ABB RobotStudio station: IRB_drawing_interface.rspag

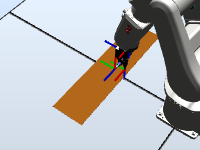
--- station ---
Station IRB_drawing_interface (saved by RobotStudio 6.7.7985.1011)
Controller IRB_120_3kg_0.58m
  mechanical unit ROB_1: IRB120_3_58__01, 6 joints, base frame (0, 0, 0) mm
Layout (positions relative to the parent item):
  - IRB120_3_58__01 [mechanism, from Robots\IRB120_3_58_G_01.rslib] at (0, 0, 0) mm; joint values [-0.0847, 0.5499, 0.7011, 0, 0.3197, 1.4861] (rad or m)
  - writing_tool_v3.1 [mechanism, from Libraries\writing_tool_v3.1.rslib] at (301.4, -25.6, 183.5) mm, rotated rx 180 ry 0 rz 90 deg
  - Cylinder_150_75_40_140_r47 [part] at (0, 0, 14) mm
  - Surface_600_150 [part]
Attachment: writing_tool_v3.1 is attached to IRB120_3_58__01 / Link6

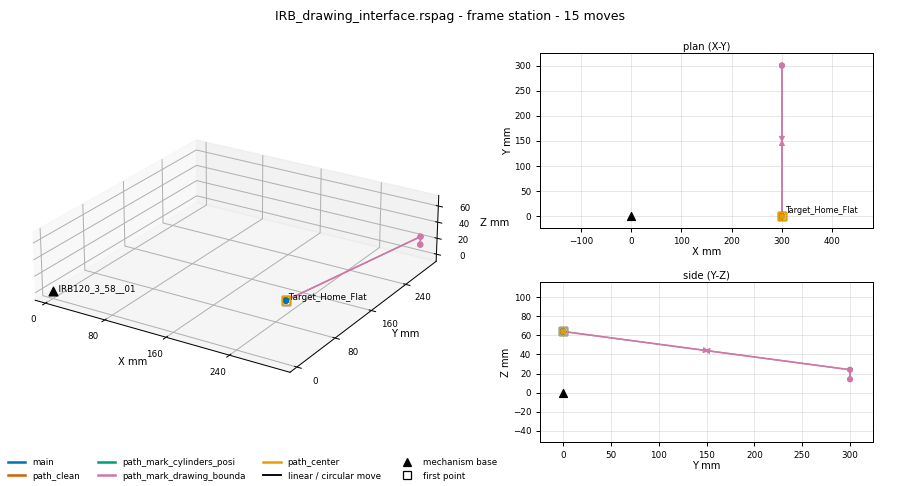
[picture p0: tool path of IRB_drawing_interface.rspag in frame station, 15 of 55 moves have a stored position in this frame; points joined in program order, loops and branches not executed]
--- Backups/IRB_120_3kg_0.58m/RAPID/TASK1/PROGMOD/Module1.mod ---
MODULE Module1

    CONST num default_flat_surface_width := 600;
    CONST num default_flat_surface_height := 150;
    CONST num default_cylinder_center_x:= 150;
    CONST num default_cylinder_center_y:=75;
    CONST num default_cylinder_bottom_height := 40;
    CONST num default_cylinder_top_height := 140;
    CONST num default_cylinder_radius := 47;

    CONST num default_cylinder_clearance := 10;
    CONST num default_cleaning_clearance := 20;

    VAR bool flag_flat:=TRUE;
    VAR bool flag_cylinder:=FALSE;
    VAR bool flag_change := TRUE;

    VAR pos message_target_pos;
    VAR intnum connectnum_pos;
    VAR string message_string;
    VAR intnum connectnum_string;

    VAR pos targetList{50000};
    VAR num targetListCount:=1;
    VAR num currentTarget:=1;

    VAR bool clean_writing_area:=FALSE;
    VAR bool stop_writing := FALSE;
    VAR bool center_the_cylinder := FALSE;
    VAR bool mark_cylinders_position := FALSE;
    VAR bool mark_drawing_boundaries := FALSE;

    VAR num flat_surface_width := default_flat_surface_width;
    VAR num flat_surface_height := default_flat_surface_height;
    VAR num cylinder_center_x:= default_cylinder_center_x;
    VAR num cylinder_center_y:=default_cylinder_center_y;
    VAR num cylinder_bottom_height := default_cylinder_bottom_height;
    VAR num cylinder_top_height := default_cylinder_top_height;
    VAR num cylinder_radius := default_cylinder_radius;
    VAR num angle;
    VAR pos flat_current_point := [0,0,47 + default_cylinder_clearance];
    VAR num cylinder_start_angle := 0;

	PERS tooldata side:=[TRUE,[[70.1,18.6,86],[0.707106781,0,0.707106781,0]],[0.4,[0,0,50],[1,0,0,0],0,0,0]];
	PERS tooldata down:=[TRUE,[[25.6,-1.4,119.5],[1,0,0,0]],[0.4,[0,0,50],[1,0,0,0],0,0,0]];
	PERS tooldata clean:=[TRUE,[[2.6,46.6,43],[0.5,-0.5,0.5,0.5]],[0.4,[0,0,50],[1,0,0,0],0,0,0]];

	PERS wobjdata WritingArea:=[FALSE,TRUE,"",[[300,300,14],[0.707,0,0,-0.707]],[[0,0,0],[1,0,0,0]]];

    CONST robtarget Target_Home_Flat:=[[300,0,50],[0,0,1,0],[0,-1,-1,0],[9E+09,9E+09,9E+09,9E+09,9E+09,9E+09]];
    VAR robtarget Target_Home_Cylinder:=[[150+default_cylinder_radius+default_cylinder_clearance,default_cylinder_center_y,default_cylinder_bottom_height],[0.707,0,-0.707,0],[0,-1,-1,0],[9E+09,9E+09,9E+09,9E+09,9E+09,9E+09]];
    CONST robtarget cleaning_target_1 := [[15,0,default_cleaning_clearance],[0,0.707,-0.707,0],[0,0,-2,1],[9E+09,9E+09,9E+09,9E+09,9E+09,9E+09]];
    CONST robtarget cleaning_target_2 := [[15,0,default_cleaning_clearance],[0,-1,.000191058,0],[0,-1,-2,1],[9E+09,9E+09,9E+09,9E+09,9E+09,9E+09]];

    PROC main()

        CONNECT connectnum_pos WITH RABMsgs_pos;
        IRMQMessage message_target_pos,connectnum_pos;
        CONNECT connectnum_string WITH RABMsgs_string;
        IRMQMessage message_string,connectnum_string;

        WHILE flag_flat=TRUE DO

            IF stop_writing THEN
                currentTarget := targetListCount;
                stop_writing := FALSE;

            ELSEIF flag_change THEN
                MoveL Target_Home_Flat,v300,z10,down\WObj:=WritingArea;
                flag_change := FALSE;

            ELSEIF clean_writing_area THEN
                path_clean;
                clean_writing_area := FALSE;

            ELSEIF center_the_cylinder THEN
                path_center;
                center_the_cylinder := FALSE;

            ELSEIF mark_cylinders_position THEN
                path_mark_cylinders_position;
                mark_cylinders_position := FALSE;

            ELSEIF mark_drawing_boundaries THEN
                path_mark_drawing_boundaries;
                mark_drawing_boundaries := FALSE;

            ELSEIF (currentTarget<>targetListCount) THEN

                targetList{currentTarget}.y:= -1 * targetList{currentTarget}.y + flat_surface_height;

                IF targetList{currentTarget}.z=0 THEN
                    MoveJ [[targetList{currentTarget}.x,targetList{currentTarget}.y,targetList{currentTarget}.z+10],[0,0,1,0],[0,-1,-1,0],[9E+09,9E+09,9E+09,9E+09,9E+09,9E+09]],v200,z10,down\WObj:=WritingArea;
                    MoveL [[targetList{currentTarget}.x,targetList{currentTarget}.y,targetList{currentTarget}.z],[0,0,1,0],[0,-1,-1,0],[9E+09,9E+09,9E+09,9E+09,9E+09,9E+09]],v300,fine,down\WObj:=WritingArea;
                ELSEIF targetList{currentTarget}.z=1 THEN
                    MoveL [[targetList{currentTarget}.x,targetList{currentTarget}.y,targetList{currentTarget}.z],[0,0,1,0],[0,-1,-1,0],[9E+09,9E+09,9E+09,9E+09,9E+09,9E+09]],v300,fine,down\WObj:=WritingArea;
                ELSEIF targetList{currentTarget}.z=2 THEN
                    MoveL [[targetList{currentTarget}.x,targetList{currentTarget}.y,targetList{currentTarget}.z],[0,0,1,0],[0,-1,-1,0],[9E+09,9E+09,9E+09,9E+09,9E+09,9E+09]],v300,fine,down\WObj:=WritingArea;
                    MoveJ [[targetList{currentTarget}.x,targetList{currentTarget}.y,targetList{currentTarget}.z+10],[0,0,1,0],[0,-1,-1,0],[9E+09,9E+09,9E+09,9E+09,9E+09,9E+09]],v200,z10,down\WObj:=WritingArea;
                ENDIF
                currentTarget:=currentTarget+1;

            ELSE
                MoveL Target_Home_Flat,v300,z10,down\WObj:=WritingArea;
            ENDIF

        ENDWHILE

        WHILE flag_cylinder=TRUE DO

            IF stop_writing THEN
                currentTarget := targetListCount;
                stop_writing := FALSE;

            ELSEIF flag_change THEN
                MoveL Target_Home_Flat,v300,z10,down\WObj:=WritingArea;
                MoveL Target_Home_Cylinder,v300,z10,side\WObj:=WritingArea;
                flag_change := FALSE;

            ELSEIF (currentTarget<>targetListCount) THEN

                targetList{currentTarget}.y:= -1 * targetList{currentTarget}.y + cylinder_top_height - cylinder_bottom_height;

                IF targetList{currentTarget}.z=0 THEN
                    curve_to_point([targetList{currentTarget}.x,targetList{currentTarget}.y, cylinder_radius + default_cylinder_clearance]);
                    curve_to_point([targetList{currentTarget}.x,targetList{currentTarget}.y, cylinder_radius]);
                ELSEIF targetList{currentTarget}.z=1 THEN
                    curve_to_point([targetList{currentTarget}.x,targetList{currentTarget}.y, cylinder_radius]);
                ELSEIF targetList{currentTarget}.z=2 THEN
                    curve_to_point([targetList{currentTarget}.x,targetList{currentTarget}.y, cylinder_radius]);
                    curve_to_point([targetList{currentTarget}.x,targetList{currentTarget}.y, cylinder_radius + default_cylinder_clearance]);
                ENDIF
                currentTarget:=currentTarget+1;

            ELSEIF clean_writing_area THEN
                !path_clean;
                clean_writing_area := FALSE;
            ELSE
                curve_to_point([0,0,cylinder_radius + default_cylinder_clearance]);
            ENDIF

        ENDWHILE

        IDelete connectnum_pos;
        IDelete connectnum_string;

    ENDPROC

    TRAP RABMsgs_pos

        VAR rmqmessage msg;
        VAR rmqheader header;
        VAR rmqslot rabclient;
        VAR num userdef;
        RMQGetMessage msg;
        RMQGetMsgHeader msg\Header:=header\SenderId:=rabclient\UserDef:=userdef;

        IF header.datatype="pos" THEN
            RMQGetMsgData msg,message_target_pos;

            targetList{targetListCount}:=message_target_pos;
            targetListCount:=targetListCount+1;

        ENDIF

    ENDTRAP

    TRAP RABMsgs_string

        VAR rmqmessage msg;
        VAR rmqheader header;
        VAR rmqslot rabclient;
        VAR num userdef;
        VAR num n;
        VAR num m;
        VAR bool convert_ok;
        RMQGetMessage msg;
        RMQGetMsgHeader msg\Header:=header\SenderId:=rabclient\UserDef:=userdef;

        IF header.datatype="string" THEN
            RMQGetMsgData msg,message_string;

            IF StrPart(message_string, 1, 4) = "func" THEN

                IF StrPart(message_string, 6, 1) = "1" THEN
                    stop_writing := TRUE;
                ELSEIF StrPart(message_string, 6, 1) = "2" THEN
                    clean_writing_area := TRUE;
                ELSEIF StrPart(message_string, 6, 1) = "3" THEN

                ELSEIF StrPart(message_string, 6, 1) = "4" THEN

                ELSEIF StrPart(message_string, 6, 1) = "5" THEN
                    center_the_cylinder := TRUE;
                ELSEIF StrPart(message_string, 6, 1) = "6" THEN
                    mark_cylinders_position := TRUE;
                ELSEIF StrPart(message_string, 6, 1) = "7" THEN
                    mark_drawing_boundaries := TRUE;
                ENDIF

            ELSEIF StrPart(message_string, 1, 4) = "para" THEN

                n := StrMatch(message_string, 1, "fsw");
                m := StrFind(message_string,n + 3,STR_WHITE);
                convert_ok := StrToVal(StrPart(message_string, n + 3, m - (n + 3)), flat_surface_width);

                n := StrMatch(message_string, 1, "fsh");
                m := StrFind(message_string,n + 3,STR_WHITE);
                convert_ok := StrToVal(StrPart(message_string, n + 3, m - (n + 3)), flat_surface_height);

                n := StrMatch(message_string, 1, "cpx");
                m := StrFind(message_string,n + 3,STR_WHITE);
                convert_ok := StrToVal(StrPart(message_string, n + 3, m - (n + 3)), cylinder_center_x);

                n := StrMatch(message_string, 1, "cpy");
                m := StrFind(message_string,n + 3,STR_WHITE);
                convert_ok := StrToVal(StrPart(message_string, n + 3, m - (n + 3)), cylinder_center_y);

                n := StrMatch(message_string, 1, "cbh");
                m := StrFind(message_string,n + 3,STR_WHITE);
                convert_ok := StrToVal(StrPart(message_string, n + 3, m - (n + 3)), cylinder_bottom_height);

                n := StrMatch(message_string, 1, "cth");
                m := StrFind(message_string,n + 3,STR_WHITE);
                convert_ok := StrToVal(StrPart(message_string, n + 3, m - (n + 3)), cylinder_top_height);

                n := StrMatch(message_string, 1, "cra");
                m := StrFind(message_string,n + 3,STR_WHITE);
                convert_ok := StrToVal(StrPart(message_string, n + 3, m - (n + 3)), cylinder_radius);

                n := StrMatch(message_string, 1, "cld");
                m := StrFind(message_string,n + 3,STR_WHITE);
                IF StrPart(message_string, n + 3, m - (n + 3)) = "True" THEN
                    flag_flat := FALSE;
                    flag_cylinder := TRUE;
                    flag_change := TRUE;
                ELSE
                    flag_flat := TRUE;
                    flag_cylinder := FALSE;
                    flag_change := TRUE;
                ENDIF

                Target_Home_Cylinder.trans := [150+cylinder_radius+default_cylinder_clearance,cylinder_center_y,cylinder_bottom_height];

            ENDIF
        ENDIF

    ENDTRAP

    PROC path_clean()
        CONST num cleaning_step := 52;
        VAR speeddata cleaning_speed := v200;
        VAR num offset_x := cleaning_step / 2;

        MoveJ Offs(Target_Home_Flat,0,0,0),cleaning_speed,z10,down\WObj:=WritingArea;
        MoveJ Offs(cleaning_target_1,cleaning_step / 2,flat_surface_height,120),cleaning_speed,z10,clean\WObj:=WritingArea;
        MoveJ Offs(cleaning_target_1,cleaning_step / 2,flat_surface_height,0),cleaning_speed,z10,clean\WObj:=WritingArea;
        FOR i FROM 0 TO 4 DO
            MoveL Offs(cleaning_target_2,offset_x,0,0),cleaning_speed,z10,clean\WObj:=WritingArea;
            offset_x:=offset_x + cleaning_step;
            MoveL Offs(cleaning_target_2,offset_x,0,0),cleaning_speed,z10,clean\WObj:=WritingArea;
            MoveL Offs(cleaning_target_1,offset_x,flat_surface_height,0),cleaning_speed,z10,clean\WObj:=WritingArea;
            IF i <> 5 THEN
                offset_x:=offset_x + cleaning_step;
                MoveL Offs(cleaning_target_1,offset_x,flat_surface_height,0),cleaning_speed,z10,clean\WObj:=WritingArea;
            ENDIF
        ENDFOR
        MoveL Offs(cleaning_target_1,0,flat_surface_height,0),cleaning_speed,z10,clean\WObj:=WritingArea;
        MoveL Offs(cleaning_target_1,0,flat_surface_height,120),cleaning_speed,z10,clean\WObj:=WritingArea;
        MoveJ Offs(Target_Home_Flat,0,0,0),cleaning_speed,z10,down\WObj:=WritingArea;
    ENDPROC

    PROC path_mark_cylinders_position()
        MoveL Target_Home_Flat,v100,fine,down\WObj:=WritingArea;
        MoveL [[cylinder_center_x+cylinder_radius*Sin(0),cylinder_center_y+cylinder_radius*Cos(0),10],[0,0,1,0],[0,-1,-1,0],[9E+09,9E+09,9E+09,9E+09,9E+09,9E+09]],v150,z0,down\WObj:=WritingArea;
        FOR i FROM 0 TO 90 DO
            MoveL [[cylinder_center_x+cylinder_radius*Sin(i*4),cylinder_center_y+cylinder_radius*Cos(i*4),0],[0,0,1,0],[0,-1,-1,0],[9E+09,9E+09,9E+09,9E+09,9E+09,9E+09]],v150,z0,down\WObj:=WritingArea;
        ENDFOR
        MoveL [[cylinder_center_x+cylinder_radius*Sin(0),cylinder_center_y+cylinder_radius*Cos(0),10],[0,0,1,0],[0,-1,-1,0],[9E+09,9E+09,9E+09,9E+09,9E+09,9E+09]],v150,z0,down\WObj:=WritingArea;
        MoveL Target_Home_Flat,v100,fine,down\WObj:=WritingArea;
    ENDPROC

    PROC path_mark_drawing_boundaries()
        MoveL Target_Home_Flat,v100,fine,down\WObj:=WritingArea;
        MoveL [[0,0,10],[0,0,1,0],[0,-1,-1,0],[9E+09,9E+09,9E+09,9E+09,9E+09,9E+09]],v150,z0,down\WObj:=WritingArea;
        MoveL [[0,0,0],[0,0,1,0],[0,-1,-1,0],[9E+09,9E+09,9E+09,9E+09,9E+09,9E+09]],v150,z0,down\WObj:=WritingArea;
        MoveL [[flat_surface_width,0,0],[0,0,1,0],[0,-1,-1,0],[9E+09,9E+09,9E+09,9E+09,9E+09,9E+09]],v150,z0,down\WObj:=WritingArea;
        MoveL [[flat_surface_width,flat_surface_height,0],[0,0,1,0],[0,-1,-1,0],[9E+09,9E+09,9E+09,9E+09,9E+09,9E+09]],v150,z0,down\WObj:=WritingArea;
        MoveL [[0,flat_surface_height,0],[0,0,1,0],[0,-1,-1,0],[9E+09,9E+09,9E+09,9E+09,9E+09,9E+09]],v150,z0,down\WObj:=WritingArea;
        MoveL [[0,0,0],[0,0,1,0],[0,-1,-1,0],[9E+09,9E+09,9E+09,9E+09,9E+09,9E+09]],v150,z0,down\WObj:=WritingArea;
        MoveL [[0,0,10],[0,0,1,0],[0,-1,-1,0],[9E+09,9E+09,9E+09,9E+09,9E+09,9E+09]],v150,z0,down\WObj:=WritingArea;
        MoveL Target_Home_Flat,v100,fine,down\WObj:=WritingArea;
    ENDPROC

    PROC path_center()
        VAR robtarget push_target;
        push_target.extax := [9E+09,9E+09,9E+09,9E+09,9E+09,9E+09];

        MoveL Target_Home_Flat,v100,fine,down\WObj:=WritingArea;

        push_target.trans := [cylinder_center_x + cylinder_radius + 30, cylinder_center_y, 100];
        push_target.rot := [0.707,0,-0.707,0];
        push_target.robconf := [0,0,0,0];
        MoveL push_target,v100,z0,clean\WObj:=WritingArea;
        push_target.trans := [cylinder_center_x + (cylinder_radius - 1.5), cylinder_center_y, 100];
        MoveL push_target,v5,fine,clean\WObj:=WritingArea;
        push_target.trans := [cylinder_center_x + cylinder_radius + 30, cylinder_center_y, 100];
        MoveL push_target,v200,z5,clean\WObj:=WritingArea;

        push_target.trans := [cylinder_center_x + cylinder_radius + 30, cylinder_center_y + cylinder_radius + 30, 100];
        push_target.rot := [0.653386,0.270345,-0.653386,0.270344];
        push_target.robconf := [0,0,-1,0];
        MoveL push_target,v200,z15,clean\WObj:=WritingArea;

        push_target.trans := [cylinder_center_x, cylinder_center_y + (cylinder_radius + 30), 100];
        push_target.rot := [0.5,0.5,-0.5,0.5];
        push_target.robconf := [0,0,-1,0];
        MoveL push_target,v100,z0,clean\WObj:=WritingArea;
        push_target.trans := [cylinder_center_x, cylinder_center_y + (cylinder_radius - 1.5), 100];
        MoveL push_target,v5,fine,clean\WObj:=WritingArea;
        push_target.trans := [cylinder_center_x, cylinder_center_y + cylinder_radius + 30, 100];
        MoveL push_target,v200,z5,clean\WObj:=WritingArea;

        push_target.trans := [cylinder_center_x - cylinder_radius - 30, cylinder_center_y + cylinder_radius + 30, 100];
        push_target.rot := [0.270311,0.6534,-0.270311,0.6534];
        push_target.robconf := [0,0,-2,0];
        MoveL push_target,v200,z15,clean\WObj:=WritingArea;

        push_target.trans := [cylinder_center_x - cylinder_radius - 30, cylinder_center_y, 100];
        push_target.rot := [0,-0.707,0,-0.707];
        push_target.robconf := [0,0,-2,0];
        MoveL push_target,v100,z0,clean\WObj:=WritingArea;
        push_target.trans := [cylinder_center_x - (cylinder_radius - 1.5), cylinder_center_y, 100];
        MoveL push_target,v5,fine,clean\WObj:=WritingArea;
        push_target.trans := [cylinder_center_x - cylinder_radius - 30, cylinder_center_y, 100];
        MoveL push_target,v200,z5,clean\WObj:=WritingArea;

        push_target.trans := [cylinder_center_x - cylinder_radius - 30, cylinder_center_y - cylinder_radius - 30, 100];
        push_target.rot := [0.271904,-0.652739,-0.271904,-0.652739];
        push_target.robconf := [0,0,-3,0];
        MoveL push_target,v200,z15,clean\WObj:=WritingArea;

        push_target.trans := [cylinder_center_x, cylinder_center_y - cylinder_radius - 30, 100];
        push_target.rot := [0.5,-0.5,-0.5,-0.5];
        push_target.robconf := [0,0,-3,0];
        MoveL push_target,v100,z0,clean\WObj:=WritingArea;
        push_target.trans := [cylinder_center_x, cylinder_center_y - (cylinder_radius - 1.5), 100];
        MoveL push_target,v5,fine,clean\WObj:=WritingArea;
        push_target.trans := [cylinder_center_x, cylinder_center_y - cylinder_radius - 30, 100];
        MoveL push_target,v200,z5,clean\WObj:=WritingArea;

        push_target.trans := [cylinder_center_x - cylinder_radius - 30, cylinder_center_y - cylinder_radius - 30, 100];
        push_target.rot := [0.271904,-0.652739,-0.271904,-0.652739];
        push_target.robconf := [0,0,-3,0];
        MoveL push_target,v200,z15,clean\WObj:=WritingArea;

        push_target.trans := [cylinder_center_x - cylinder_radius - 30, cylinder_center_y + cylinder_radius + 30, 100];
        push_target.rot := [0.270311,0.6534,-0.270311,0.6534];
        push_target.robconf := [0,0,-2,0];
        MoveL push_target,v200,z15,clean\WObj:=WritingArea;

        push_target.trans := [cylinder_center_x + cylinder_radius + 30, cylinder_center_y + cylinder_radius + 30, 100];
        push_target.rot := [0.653386,0.270345,-0.653386,0.270344];
        push_target.robconf := [0,0,-1,0];
        MoveL push_target,v200,z15,clean\WObj:=WritingArea;

        MoveL Target_Home_Flat,v100,fine,down\WObj:=WritingArea;

    ENDPROC

    PROC curve_to_point(pos flat_next_point)
        VAR num flat_distance_between_points;
        VAR num flat_delta_x;
        VAR num flat_delta_y;
        VAR num flat_next_x;
        VAR num flat_next_y;
        VAR pos generated_point;
        VAR orient cylinder_tool_orientation := [0.707,0,0.707,0];
        VAR confdata cylinder_tool_conf := [0,0,0,0];

        flat_delta_x := flat_next_point.x - flat_current_point.x;
        flat_delta_y := flat_next_point.y - flat_current_point.y;
        flat_distance_between_points := Round(Sqrt(Pow(flat_delta_x, 2) + Pow(flat_delta_y, 2)));

        IF flat_distance_between_points <> 0 THEN
            FOR i FROM 0 TO flat_distance_between_points DO
                flat_next_x := flat_current_point.x + (flat_delta_x / flat_distance_between_points) * i;
                flat_next_y := flat_current_point.y + (flat_delta_y / flat_distance_between_points) * i;

                angle := flat_next_x * 180 / (cylinder_radius * pi) + cylinder_start_angle;

                IF angle <= 90 THEN
                    cylinder_tool_conf := [0,-1,-1,0];
                ELSEIF angle <= 180 THEN
                    cylinder_tool_conf := [0,-1,-2,0];
                ELSEIF angle <= 270 THEN
                    cylinder_tool_conf := [0,-1,-3,0];
                ELSEIF angle <= 360 THEN
                    cylinder_tool_conf := [0,-1,-4,0];
                ENDIF

                generated_point.x := flat_next_point.z * Cos(angle) + cylinder_center_x;
                generated_point.y := flat_next_point.z * Sin(angle) + cylinder_center_y;
                generated_point.z := flat_next_y + cylinder_bottom_height;
                cylinder_tool_orientation := OrientZYX(angle, -90, 0);
                MoveL [generated_point,cylinder_tool_orientation,cylinder_tool_conf,[9E+09,9E+09,9E+09,9E+09,9E+09,9E+09]],v50,z0,side\WObj:=WritingArea;
            ENDFOR
        ELSE
            flat_next_x := flat_current_point.x + flat_delta_x;
            flat_next_y := flat_current_point.y + flat_delta_y;

            angle := flat_next_x * 180 / (cylinder_radius * pi) + cylinder_start_angle;

            IF angle <= 90 THEN
                cylinder_tool_conf := [0,-1,-1,0];
            ELSEIF angle <= 180 THEN
                cylinder_tool_conf := [0,-1,-2,0];
            ELSEIF angle <= 270 THEN
                cylinder_tool_conf := [0,-1,-3,0];
            ELSEIF angle <= 360 THEN
                cylinder_tool_conf := [0,-1,-4,0];
            ELSEIF angle <= 450 THEN
                cylinder_tool_conf := [0,-1,-5,0];
            ENDIF

            generated_point.x := flat_next_point.z * Cos(angle) + cylinder_center_x;
            generated_point.y := flat_next_point.z * Sin(angle) + cylinder_center_y;
            generated_point.z := flat_next_y + cylinder_bottom_height;
            cylinder_tool_orientation := OrientZYX(angle, -90, 0);
            MoveL [generated_point,cylinder_tool_orientation,cylinder_tool_conf,[9E+09,9E+09,9E+09,9E+09,9E+09,9E+09]],v10,fine,side\WObj:=WritingArea;
        ENDIF
        flat_current_point := flat_next_point;
    ENDPROC

ENDMODULE
